Staubli VAL3: robotStateInq.pgx

public program robotStateInq(pointRx& x_pPoint_Pos[], num& x_nPoint_Vel[], num& x_nPoint_Accel[], jointRx& x_jJoint_Pos[], num& x_nJoint_Vel[], num& x_nJoint_Accel[], num& x_nVel[])
  local num l_nJoint_Vel[6]
  local num l_nNum
  local num l_nPoint_Vel[6]
begin

  //==================== 获取机器人执行当前指令过程中的运动状态（位置，速度，加速度(Cartesian/Joint Space)）（注意单位换算） ====================

  //---------- 获取机器人笛卡尔空间（Cartersian Space）下的运动状态 ----------
  //应确定4ms末机器人的状态，但是4ms很短，获取中间的状态影响不大，但应尽量接近4ms末
  //delay(0.003)

  //获取机器人的位置和姿态（实时从编码器测量得来）（单位：mm,°）
  x_pPoint_Pos=$getPosFbk(flange,world)

  //获取机器人的速度（平移+旋转）（单位：mm/s,°/s）
  x_nVel=$getSpeedFbk(flange,world,l_nPoint_Vel[0],l_nPoint_Vel[1],l_nPoint_Vel[2],l_nPoint_Vel[3],l_nPoint_Vel[4],l_nPoint_Vel[5])

  //获取（差分计算）机器人的加速度（平移+旋转）（（当前机器人笛卡尔-上一次机器人笛卡尔速度）/循环时间）（单位：mm/s^2,°/s^2）
  for l_nNum=0 to 5
    x_nPoint_Accel[l_nNum]=(l_nPoint_Vel[l_nNum]-nNowPointVel[l_nNum])/0.004
    x_nPoint_Vel[l_nNum]=l_nPoint_Vel[l_nNum]
  endFor


  //---------- 获取机器人关节空间（Joint Space）下的运动状态 ----------
  //获得机器人的关节位置（实时从编码器测量得来）（单位：°）
  x_jJoint_Pos=$getJntFbk()

  //获取机器人的关节速度（单位：°/s）
  $getJntSpeedFbk(l_nJoint_Vel)

  //获取（差分计算）机器人的关节加速度（（当前机器人关节速度-上一次机器人关节速度）/循环时间）（单位：°/s^2）
  for l_nNum=0 to 5
    x_nJoint_Accel[l_nNum]=(l_nJoint_Vel[l_nNum]-nNowJointVel[l_nNum])/0.004
    x_nJoint_Vel[l_nNum]=l_nJoint_Vel[l_nNum]
  endFor

end
